Fanuc KAREL source: kb00187.KL

-- PROVISIONAL review KL for V1013-1; original PC SHA256 7a02f3a0da78108d7505fe69981af9a2a921f0a31e0281e6ec3b71899e2c5177
-- Incomplete behavior may be omitted. Consult companion uncertainty JSON. Do not deploy.
PROGRAM KB00187
%NOLOCKGROUP
VAR
  P1 : REAL
  RESULT : REAL
BEGIN
  -- UNRESOLVED_PC offsets 5-16; opcodes 2E,23
  -- UNRESOLVED_PC offsets 21-36; opcodes 27,22,76,23
  -- UNRESOLVED_PC offsets 41-45; opcodes 7F
END KB00187
